TYPE ST_PERSISTENCY_OUT :
STRUCT
	busy:					BOOL;
	error:					BOOL;
	beckhoffErrorId:		UDINT;
	errorIdEnum:			E_ADS_ERRORS;
END_STRUCT
END_TYPE

(* stored: Version 1.1.0.1, ProductVersion 3.1.4026.18
   DUT ST_PERSISTENCY_OUT: Id {390c118b-8cad-417b-a2ec-244ce6c799bb} *)
